# EPICS substitutions: apps/CaenHVApp/Db/CaenHV_crate2.substitutions
file "db/AS503_Chan.template" {
pattern
    {P,      H,  S,   V}
    {hchv,   2,  00,  000}
    {hchv,   2,  00,  001}
    {hchv,   2,  00,  002}
    {hchv,   2,  00,  003}
    {hchv,   2,  00,  004}
    {hchv,   2,  00,  005}
    {hchv,   2,  00,  006}
    {hchv,   2,  00,  007}
    {hchv,   2,  00,  008}
    {hchv,   2,  00,  009}
    {hchv,   2,  00,  010}
    {hchv,   2,  00,  011}
    {hchv,   2,  00,  012}
    {hchv,   2,  00,  013}
    {hchv,   2,  00,  014}
    {hchv,   2,  00,  015}
}
file "db/AS503_Chan.template" {
pattern
    {P,      H,  S,   V}
    {hchv,   2,  01, 000}
    {hchv,   2,  01, 001}
    {hchv,   2,  01, 002}
    {hchv,   2,  01, 003}
    {hchv,   2,  01, 004}
    {hchv,   2,  01, 005}
    {hchv,   2,  01, 006}
    {hchv,   2,  01, 007}
    {hchv,   2,  01, 008}
    {hchv,   2,  01, 009}
    {hchv,   2,  01, 010}
    {hchv,   2,  01, 011}
    {hchv,   2,  01, 012}
    {hchv,   2,  01, 013}
    {hchv,   2,  01, 014}
    {hchv,   2,  01, 015}
}
file "db/AS503_Chan.template" {
pattern
    {P,      H,  S,   V}
    {hchv,   2,  02, 000}
    {hchv,   2,  02, 001}
    {hchv,   2,  02, 002}
    {hchv,   2,  02, 003}
    {hchv,   2,  02, 004}
    {hchv,   2,  02, 005}
    {hchv,   2,  02, 006}
    {hchv,   2,  02, 007}
    {hchv,   2,  02, 008}
    {hchv,   2,  02, 009}
    {hchv,   2,  02, 010}
    {hchv,   2,  02, 011}
    {hchv,   2,  02, 012}
    {hchv,   2,  02, 013}
    {hchv,   2,  02, 014}
    {hchv,   2,  02, 015}
}
file "db/AS503_Chan.template" {
pattern
    {P,      H,  S,   V}
    {hchv,   2,  03, 000}
    {hchv,   2,  03, 001}
    {hchv,   2,  03, 002}
    {hchv,   2,  03, 003}
    {hchv,   2,  03, 004}
    {hchv,   2,  03, 005}
    {hchv,   2,  03, 006}
    {hchv,   2,  03, 007}
    {hchv,   2,  03, 008}
    {hchv,   2,  03, 009}
    {hchv,   2,  03, 010}
    {hchv,   2,  03, 011}
    {hchv,   2,  03, 012}
    {hchv,   2,  03, 013}
    {hchv,   2,  03, 014}
    {hchv,   2,  03, 015}
}
